(* IEC 61131-3 sources: RAG_PLC/data/result/test/033, 2 files *)

(* ---- wrapped.st ---- *)
(* =========================================================
   Generated by PLC-Eval Benchmark Wrapper
   ========================================================= *)

FUNCTION_BLOCK LLM_Wrapper_FB
VAR_INPUT
	LTIME : UDINT;
	DST : BOOL;
	TIME_ZONE_OFFSET : INT;
END_VAR

VAR_OUTPUT
	UTC : UDINT;
END_VAR

UTC := LTIME + _INT_TO_UDINT(TIME_ZONE_OFFSET * 60);
IF DST THEN UTC := UTC + UDINT#3600; END_IF;
END_FUNCTION_BLOCK

PROGRAM Auto_Proxy_Prg
  VAR
    instance : LLM_Wrapper_FB;
  END_VAR

  instance();
END_PROGRAM

CONFIGURATION Config0
  RESOURCE Res0 ON PLC
    TASK TaskMain(INTERVAL := T#20ms, PRIORITY := 0);
    PROGRAM Inst0 WITH TaskMain : Auto_Proxy_Prg;
  END_RESOURCE
END_CONFIGURATION

(* ---- raw_code.st ---- *)
VAR_INPUT
	LTIME : UDINT;
	DST : BOOL;
	TIME_ZONE_OFFSET : INT;
END_VAR

VAR_OUTPUT
	UTC : UDINT;
END_VAR

UTC := LTIME + _INT_TO_UDINT(TIME_ZONE_OFFSET * 60);
IF DST THEN UTC := UTC + UDINT#3600; END_IF;
